Fanuc KAREL source: test_files.kl

PROGRAM test_files
%NOLOCKGROUP

%include systemlib.codes.klt
%include systemlib.datatypes.klt

VAR
  testFL : FILE

%include kunit.klh
%include strings.klh
%include files.klh

BEGIN

  kunit_done
END test_files
